Fanuc KAREL source: kc00037.KL

-- PROVISIONAL review KL for V1013-1; original PC SHA256 ad3884b45906132154ba3184631f64179827c4045ac6e7ac960b4e549d3cff0f
-- Incomplete behavior may be omitted. Consult companion uncertainty JSON. Do not deploy.
PROGRAM KC00037
%NOLOCKGROUP
BEGIN
  -- UNRESOLVED_PC offsets 5-29; opcodes 27,22,2A,22,22,31
  -- UNRESOLVED_PC offsets 34-38; opcodes 7F
END KC00037
